FUNCTION CheckLRangeUnsigned : ULINT
VAR_INPUT
	value, lower, upper: ULINT;
END_VAR

{noflow}

IF (value < lower) THEN
	CheckLRangeUnsigned := lower;
	oaksGVL.udiCheckLRangeUnsigned := oaksGVL.udiCheckLRangeUnsigned + 1;
ELSIF(value > upper) THEN
	CheckLRangeUnsigned := upper;
	oaksGVL.udiCheckLRangeUnsigned := oaksGVL.udiCheckLRangeUnsigned + 1;
ELSE
	CheckLRangeUnsigned := value;
END_IF
{flow}

END_FUNCTION

(* stored: Version 1.1.0.1, ProductVersion 3.1.4022.18
   POU CheckLRangeUnsigned: Id {d74201ea-6ab8-4448-94d8-46eeeb4e6816}, SpecialFunc CheckLRangeUnsigned *)
